TYPE ST_UserControl_Manual_Cylinder_ToHmi :
STRUCT
	bVisible : BOOL;
	stObjectName				: ST_Text;
	stButton_Hp,
	stButton_Mp,
	stButton_Wp	: ST_HMI_BUTTON_OUT;
	bVisible_Button_Mp			: bool;
END_STRUCT
END_TYPE

(* stored: Version 1.1.0.1, ProductVersion 3.1.4024.11
   DUT ST_UserControl_Manual_Cylinder_ToHmi: Id {9168cae2-ba6a-403f-9d39-a1833c7e53a4} *)
